FUNCTION FC_FilePathGenerator : T_MaxString
VAR_INPUT
	iPath:			T_MaxString;
	iFile:			T_MaxString;
END_VAR

FC_FilePathGenerator := FC_3strConcat(iStr1 := iPath, iStr2 := IING.STRING_BACKSLASH, iStr3 := iFile);

END_FUNCTION

(* stored: Version 1.1.0.1, ProductVersion 3.1.4026.18
   POU FC_FilePathGenerator: Id {063c12d0-8836-4cce-adee-4e73ee1cd8a6}, SpecialFunc None *)
